FUNCTION_BLOCK FB_LamparaTemporizada_IL_2
// Lampara temporizada con tiempo de espera prolongado
VAR_INPUT
    TiempoEncendido   : TIME := T#2S;
END_VAR
VAR_OUTPUT
    TiempoPendiente   : TIME;
END_VAR
VAR
    Temporizador      : TON;
    Lampara   AT %Q*  : BOOL;
    Pulsador  AT %I*  : BOOL;
END_VAR

// NETWORK 1
// instruction list
CAL     Temporizador(
    IN      := NOT Pulsador AND Lampara,
    PT      := TiempoEncendido)

// NETWORK 2
// instruction list
LD      TiempoEncendido
SUB     Temporizador.ET
ST      TiempoPendiente

// NETWORK 3
// instruction list
LD      Pulsador
S       Lampara

// NETWORK 4
// instruction list
LD      Temporizador.Q
R       Lampara

// NETWORK 5

END_FUNCTION_BLOCK

(* stored: Version 1.1.0.1, ProductVersion 3.1.4024.15
   POU FB_LamparaTemporizada_IL_2: Id {90ff3b62-3fc7-4d62-b126-c7ec81dbfcb9}, SpecialFunc None *)
